{attribute addProperty BoxType "EL3681-0000-0017"}
{attribute addProperty Id "SAI_InputsAT %I*SAI_Inputs_C1A1928F4860SAI_RangeAT %I*SAI_Range_BF31F39A1620SAI_Range_1AT %Q*SAI_Range_E3AE57CD1620WcStateAT %I*WcState_F855686C1620InfoDataAT %I*InfoData_BC63D37F80100"}
{attribute addProperty CRC "1598998197"}
{attribute addProperty SizeInBites "176"}
{attribute addProperty SizeInBytes "22"}
TYPE EL3681_494E7C6C :
STRUCT
	{attribute addProperty Name "SAI_Inputs"}
	SAI_Inputs : SAI_Inputs_C1A1928F;
	{attribute addProperty Name "SAI_Range"}
	SAI_Range : SAI_Range_BF31F39A;
	{attribute addProperty Name "SAI_Range_1"}
	SAI_Range_1 : SAI_Range_E3AE57CD;
	{attribute addProperty Name "WcState"}
	WcState : WcState_F855686C;
	{attribute addProperty Name "InfoData"}
	InfoData : InfoData_BC63D37F;
END_STRUCT
END_TYPE

(* stored: Version 1.2.0.0, ProductVersion 3.1.4024.9
   DUT EL3681_494E7C6C: Id {7d1e55b3-ddfb-4f39-a194-9007c9ed57aa} *)
